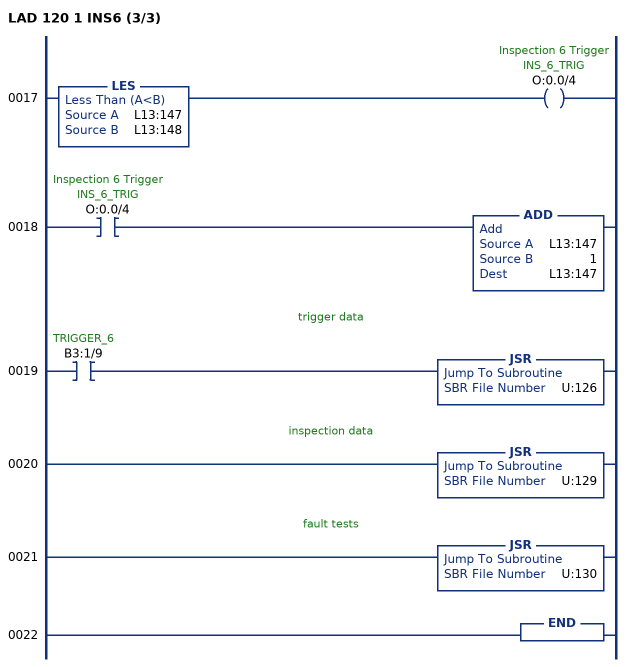
% Rung: 17 %
SOR LES L13:147 L13:148 OTE O:0.0/4 EOR
%   O:0.0/4  INS_6_TRIG  "Inspection 6 Trigger" %
% Rung: 18 %
SOR XIC O:0.0/4 ADD L13:147 1 L13:147 EOR
%   O:0.0/4  INS_6_TRIG  "Inspection 6 Trigger" %
% Rung: 19 %
% trigger data %
SOR XIC B3:1/9 JSR U:126 EOR
%   B3:1/9  TRIGGER_6 %
% Rung: 20 %
% inspection data %
SOR JSR U:129 EOR
% Rung: 21 %
% fault tests %
SOR JSR U:130 EOR
% Rung: 22 %
SOR END EOR

LADDER 121 "2 INS6RESU"
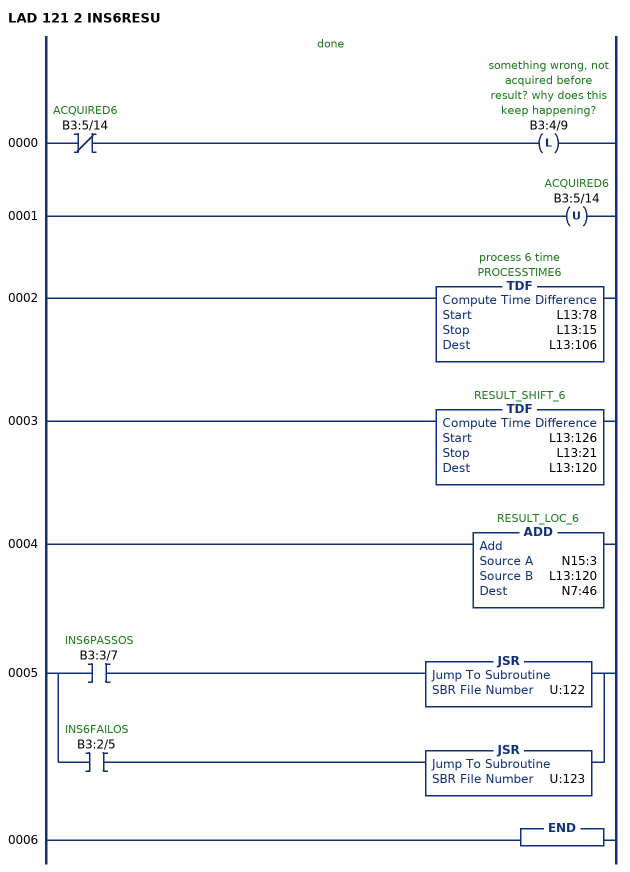
% Rung: 0 %
% done %
SOR XIO B3:5/14 OTL B3:4/9 EOR
%   B3:5/14  ACQUIRED6 %
%   B3:4/9  "something wrong, not acquired before result? why does this keep happening?" %
% Rung: 1 %
SOR OTU B3:5/14 EOR
%   B3:5/14  ACQUIRED6 %
% Rung: 2 %
SOR TDF L13:78 L13:15 L13:106 EOR
%   L13:78  TIMEOFACQ6  "the time of the last acquire" %
%   L13:15  THE_TIME %
%   L13:106  PROCESSTIME6  "process 6 time" %
% Rung: 3 %
SOR TDF L13:126 L13:21 L13:120 EOR
%   L13:126  PROCESS_START_POS_6 %
%   L13:21  TOP_POSITION %
%   L13:120  RESULT_SHIFT_6 %
% Rung: 4 %
SOR ADD N15:3 L13:120 N7:46 EOR
%   N15:3  INS_6_TRIG_LOC %
%   L13:120  RESULT_SHIFT_6 %
%   N7:46  RESULT_LOC_6 %
% Rung: 5 %
SOR BST XIC B3:3/7 JSR U:122 NXB XIC B3:2/5 JSR U:123 BND EOR
%   B3:3/7  INS6PASSOS %
%   B3:2/5  INS6FAILOS %
% Rung: 6 %
SOR END EOR

LADDER 122 "3 INS6PASS"
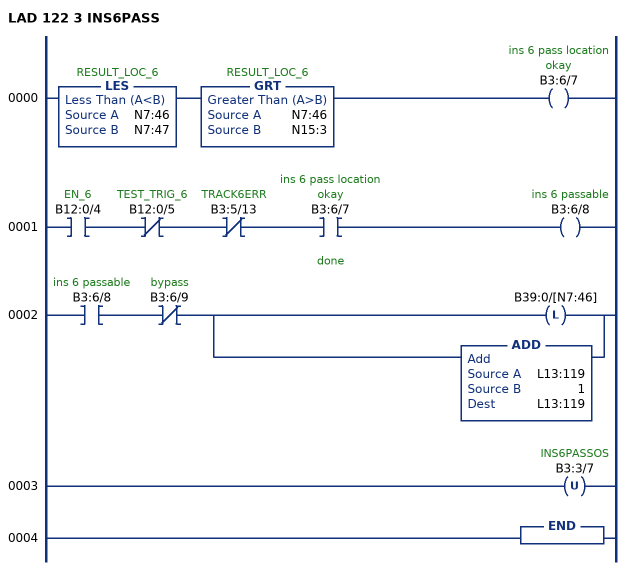
% Rung: 0 %
SOR LES N7:46 N7:47 GRT N7:46 N15:3 OTE B3:6/7 EOR
%   N7:46  RESULT_LOC_6 %
%   N7:47  INS6_MAX_SHIFT  "ins 6 maximum result location" %
%   N15:3  INS_6_TRIG_LOC %
%   B3:6/7  "ins 6 pass location okay" %
% Rung: 1 %
SOR XIC B12:0/4 XIO B12:0/5 XIO B3:5/13 XIC B3:6/7 OTE B3:6/8 EOR
%   B12:0/4  EN_6 %
%   B12:0/5  TEST_TRIG_6 %
%   B3:5/13  TRACK6ERR %
%   B3:6/7  "ins 6 pass location okay" %
%   B3:6/8  "ins 6 passable" %
% Rung: 2 %
% done %
SOR XIC B3:6/8 XIO B3:6/9 BST OTL B39:0/[N7:46] NXB ADD L13:119 1 L13:119 BND EOR
%   B3:6/8  "ins 6 passable" %
%   B3:6/9  "bypass" %
%   N7:46  RESULT_LOC_6 %
% Rung: 3 %
SOR OTU B3:3/7 EOR
%   B3:3/7  INS6PASSOS %
% Rung: 4 %
SOR END EOR

LADDER 123 "4 INS6FAIL"
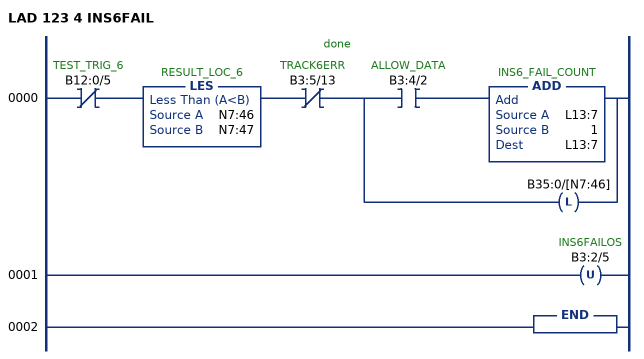
% Rung: 0 %
% done %
SOR XIO B12:0/5 LES N7:46 N7:47 XIO B3:5/13 BST XIC B3:4/2 ADD L13:7 1 L13:7 NXB OTL B35:0/[N7:46] BND EOR
%   B12:0/5  TEST_TRIG_6 %
%   N7:46  RESULT_LOC_6 %
%   N7:47  INS6_MAX_SHIFT  "ins 6 maximum result location" %
%   B3:5/13  TRACK6ERR %
%   B3:4/2  ALLOW_DATA %
%   L13:7  INS6_FAIL_COUNT %
%   B35:0  TOP_NG %
% Rung: 1 %
SOR OTU B3:2/5 EOR
%   B3:2/5  INS6FAILOS %
% Rung: 2 %
SOR END EOR

LADDER 124 "5 INS6ACQ"
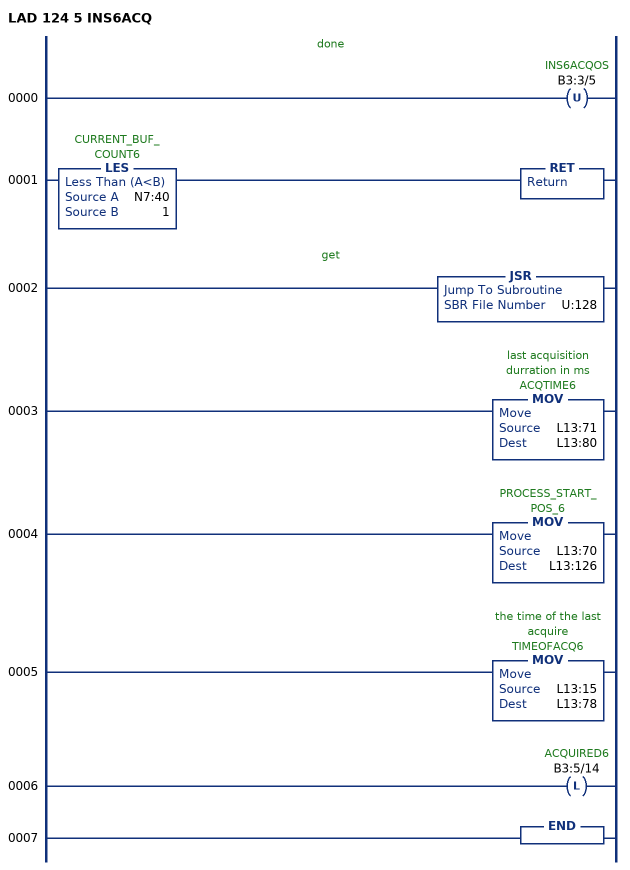
% Rung: 0 %
% done %
SOR OTU B3:3/5 EOR
%   B3:3/5  INS6ACQOS %
% Rung: 1 %
SOR LES N7:40 1 RET EOR
%   N7:40  CURRENT_BUF_COUNT6 %
% Rung: 2 %
% get %
SOR JSR U:128 EOR
% Rung: 3 %
SOR MOV L13:71 L13:80 EOR
%   L13:71  TIME_SPAN6 %
%   L13:80  ACQTIME6  "last acquisition durration in ms" %
% Rung: 4 %
SOR MOV L13:70 L13:126 EOR
%   L13:70  PULLED_POSITION6 %
%   L13:126  PROCESS_START_POS_6 %
% Rung: 5 %
SOR MOV L13:15 L13:78 EOR
%   L13:15  THE_TIME %
%   L13:78  TIMEOFACQ6  "the time of the last acquire" %
% Rung: 6 %
SOR OTL B3:5/14 EOR
%   B3:5/14  ACQUIRED6 %
% Rung: 7 %
SOR END EOR

LADDER 125 "6 Q6TESTTR"
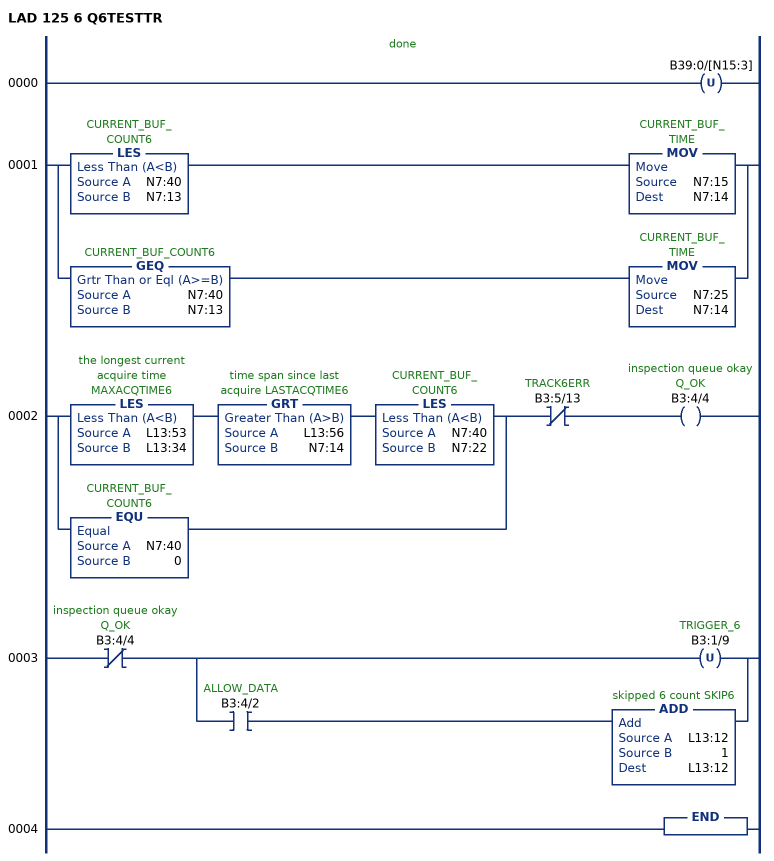
% Rung: 0 %
% done %
SOR OTU B39:0/[N15:3] EOR
%   N15:3  INS_6_TRIG_LOC %
% Rung: 1 %
SOR BST LES N7:40 N7:13 MOV N7:15 N7:14 NXB GEQ N7:40 N7:13 MOV N7:25 N7:14 BND EOR
%   N7:40  CURRENT_BUF_COUNT6 %
%   N7:13  BUF_TRANS  "cam to pc buf transition" %
%   N7:15  CAM_BUF_TIME  "cam buf time" %
%   N7:14  CURRENT_BUF_TIME %
%   N7:25  PC_BUF_TIME  "pc buf time" %
% Rung: 2 %
SOR BST LES L13:53 L13:34 GRT L13:56 N7:14 LES N7:40 N7:22 NXB EQU N7:40 0 BND XIO B3:5/13 OTE B3:4/4 EOR
%   L13:53  MAXACQTIME6  "the longest current acquire time" %
%   L13:34  MAX_ACQ_ALL  "absolute max acquire time before bypass trigger" %
%   L13:56  LASTACQTIME6  "time span since last acquire" %
%   N7:14  CURRENT_BUF_TIME %
%   N7:40  CURRENT_BUF_COUNT6 %
%   N7:22  MAX_BUF_ALL  "max buffer count alowed before bypass" %
%   B3:5/13  TRACK6ERR %
%   B3:4/4  Q_OK  "inspection queue okay" %
% Rung: 3 %
SOR XIO B3:4/4 BST OTU B3:1/9 NXB XIC B3:4/2 ADD L13:12 1 L13:12 BND EOR
%   B3:4/4  Q_OK  "inspection queue okay" %
%   B3:1/9  TRIGGER_6 %
%   B3:4/2  ALLOW_DATA %
%   L13:12  SKIP6  "skipped 6 count" %
% Rung: 4 %
SOR END EOR

LADDER 126 "7 INS6TRIG"
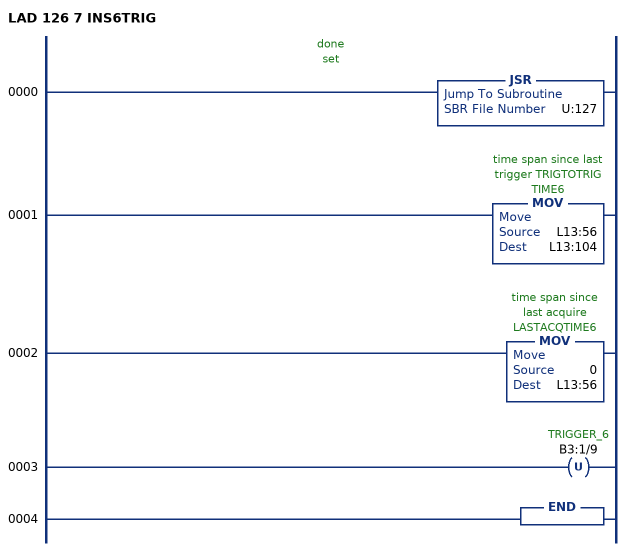
% Rung: 0 %
% done
% set %
SOR JSR U:127 EOR
% Rung: 1 %
SOR MOV L13:56 L13:104 EOR
%   L13:56  LASTACQTIME6  "time span since last acquire" %
%   L13:104  TRIGTOTRIGTIME6  "time span since last trigger" %
% Rung: 2 %
SOR MOV 0 L13:56 EOR
%   L13:56  LASTACQTIME6  "time span since last acquire" %
% Rung: 3 %
SOR OTU B3:1/9 EOR
%   B3:1/9  TRIGGER_6 %
% Rung: 4 %
SOR END EOR

LADDER 127 "8 FIFO6SET"
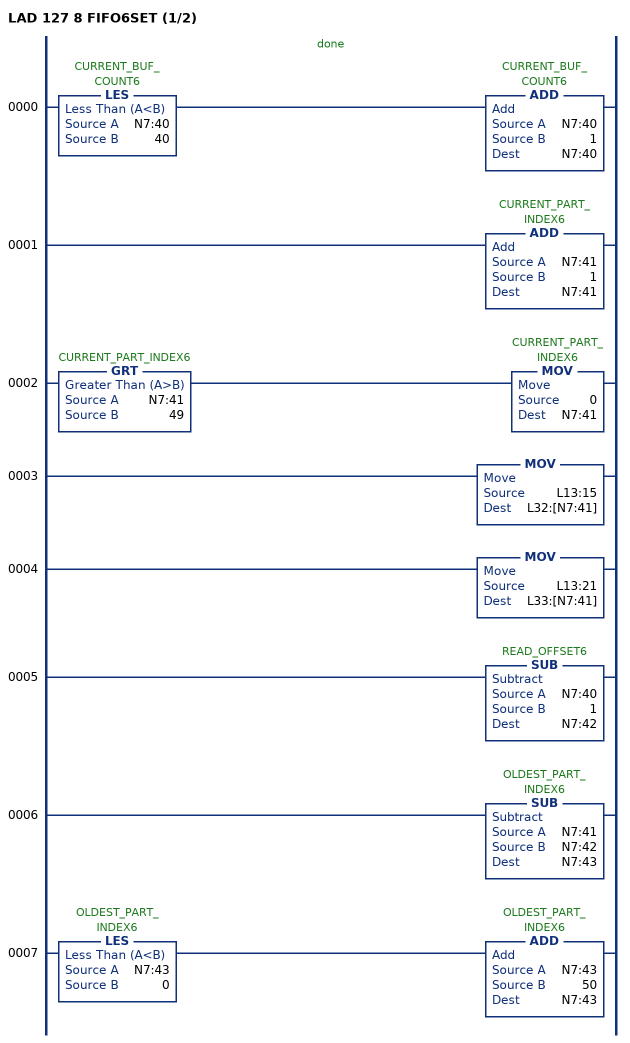
% Rung: 0 %
% done %
SOR LES N7:40 40 ADD N7:40 1 N7:40 EOR
%   N7:40  CURRENT_BUF_COUNT6 %
% Rung: 1 %
SOR ADD N7:41 1 N7:41 EOR
%   N7:41  CURRENT_PART_INDEX6 %
% Rung: 2 %
SOR GRT N7:41 49 MOV 0 N7:41 EOR
%   N7:41  CURRENT_PART_INDEX6 %
% Rung: 3 %
SOR MOV L13:15 L32:[N7:41] EOR
%   L13:15  THE_TIME %
%   N7:41  CURRENT_PART_INDEX6 %
% Rung: 4 %
SOR MOV L13:21 L33:[N7:41] EOR
%   L13:21  TOP_POSITION %
%   N7:41  CURRENT_PART_INDEX6 %
% Rung: 5 %
SOR SUB N7:40 1 N7:42 EOR
%   N7:40  CURRENT_BUF_COUNT6 %
%   N7:42  READ_OFFSET6 %
% Rung: 6 %
SOR SUB N7:41 N7:42 N7:43 EOR
%   N7:41  CURRENT_PART_INDEX6 %
%   N7:42  READ_OFFSET6 %
%   N7:43  OLDEST_PART_INDEX6 %
% Rung: 7 %
SOR LES N7:43 0 ADD N7:43 50 N7:43 EOR
%   N7:43  OLDEST_PART_INDEX6 %

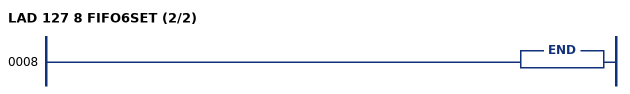
% Rung: 8 %
SOR END EOR

LADDER 128 "9 FIFO6GET"
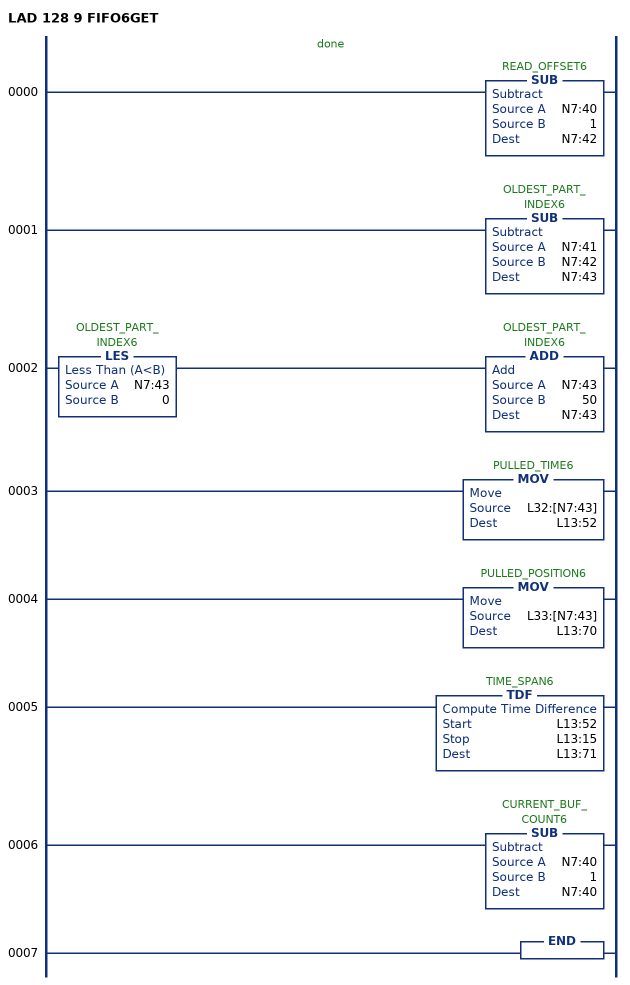
% Rung: 0 %
% done %
SOR SUB N7:40 1 N7:42 EOR
%   N7:40  CURRENT_BUF_COUNT6 %
%   N7:42  READ_OFFSET6 %
% Rung: 1 %
SOR SUB N7:41 N7:42 N7:43 EOR
%   N7:41  CURRENT_PART_INDEX6 %
%   N7:42  READ_OFFSET6 %
%   N7:43  OLDEST_PART_INDEX6 %
% Rung: 2 %
SOR LES N7:43 0 ADD N7:43 50 N7:43 EOR
%   N7:43  OLDEST_PART_INDEX6 %
% Rung: 3 %
SOR MOV L32:[N7:43] L13:52 EOR
%   N7:43  OLDEST_PART_INDEX6 %
%   L13:52  PULLED_TIME6 %
% Rung: 4 %
SOR MOV L33:[N7:43] L13:70 EOR
%   N7:43  OLDEST_PART_INDEX6 %
%   L13:70  PULLED_POSITION6 %
% Rung: 5 %
SOR TDF L13:52 L13:15 L13:71 EOR
%   L13:52  PULLED_TIME6 %
%   L13:15  THE_TIME %
%   L13:71  TIME_SPAN6 %
% Rung: 6 %
SOR SUB N7:40 1 N7:40 EOR
%   N7:40  CURRENT_BUF_COUNT6 %
% Rung: 7 %
SOR END EOR

LADDER 129 "10INSDATA6"
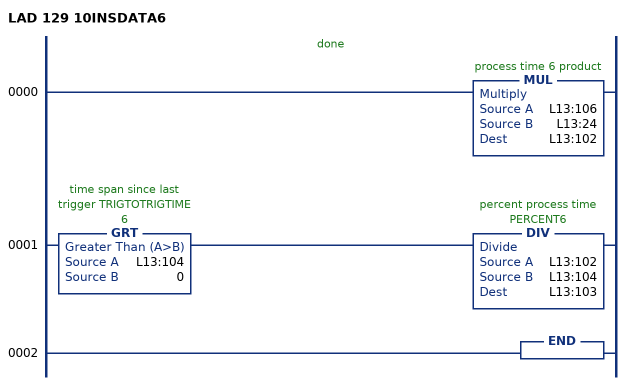
% Rung: 0 %
% done %
SOR MUL L13:106 L13:24 L13:102 EOR
%   L13:106  PROCESSTIME6  "process 6 time" %
%   L13:24  "multiplyer to make devision come out to a percentage" %
%   L13:102  "process time 6 product" %
% Rung: 1 %
SOR GRT L13:104 0 DIV L13:102 L13:104 L13:103 EOR
%   L13:104  TRIGTOTRIGTIME6  "time span since last trigger" %
%   L13:102  "process time 6 product" %
%   L13:103  PERCENT6  "percent process time" %
% Rung: 2 %
SOR END EOR

LADDER 130 "11TSTFALT6"
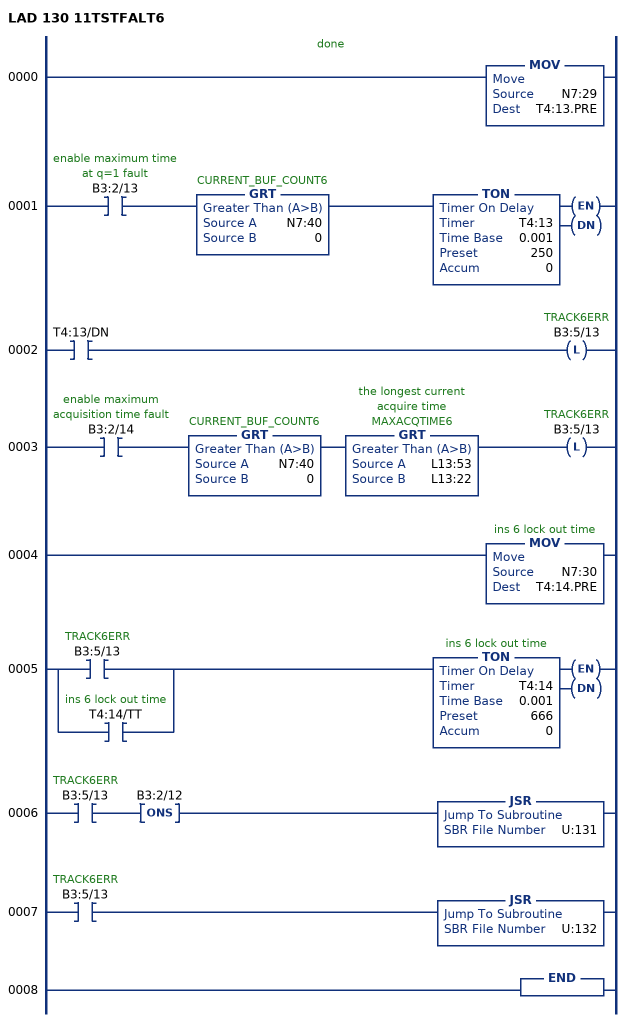
% Rung: 0 %
% done %
SOR MOV N7:29 T4:13.PRE EOR
%   N7:29  "max allowed ms time for q to be above 1 if safe fault is used" %
% Rung: 1 %
SOR XIC B3:2/13 GRT N7:40 0 TON T4:13 0.001 250 0 EOR
%   B3:2/13  "enable maximum time at q=1 fault" %
%   N7:40  CURRENT_BUF_COUNT6 %
% Rung: 2 %
SOR XIC T4:13/DN OTL B3:5/13 EOR
%   B3:5/13  TRACK6ERR %
% Rung: 3 %
SOR XIC B3:2/14 GRT N7:40 0 GRT L13:53 L13:22 OTL B3:5/13 EOR
%   B3:2/14  "enable maximum acquisition time fault" %
%   N7:40  CURRENT_BUF_COUNT6 %
%   L13:53  MAXACQTIME6  "the longest current acquire time" %
%   L13:22  "maximum of the longest acquire time allowed if maximum acquire time fault is enabled" %
%   B3:5/13  TRACK6ERR %
% Rung: 4 %
SOR MOV N7:30 T4:14.PRE EOR
%   N7:30  "ms time setting to lock out inspection to give all pending images a chance to clear" %
%   T4:14  "ins 6 lock out time" %
% Rung: 5 %
SOR BST XIC B3:5/13 NXB XIC T4:14/TT BND TON T4:14 0.001 666 0 EOR
%   B3:5/13  TRACK6ERR %
%   T4:14  "ins 6 lock out time" %
% Rung: 6 %
SOR XIC B3:5/13 ONS B3:2/12 JSR U:131 EOR
%   B3:5/13  TRACK6ERR %
% Rung: 7 %
SOR XIC B3:5/13 JSR U:132 EOR
%   B3:5/13  TRACK6ERR %
% Rung: 8 %
SOR END EOR

LADDER 131 "12INS6FIX1"
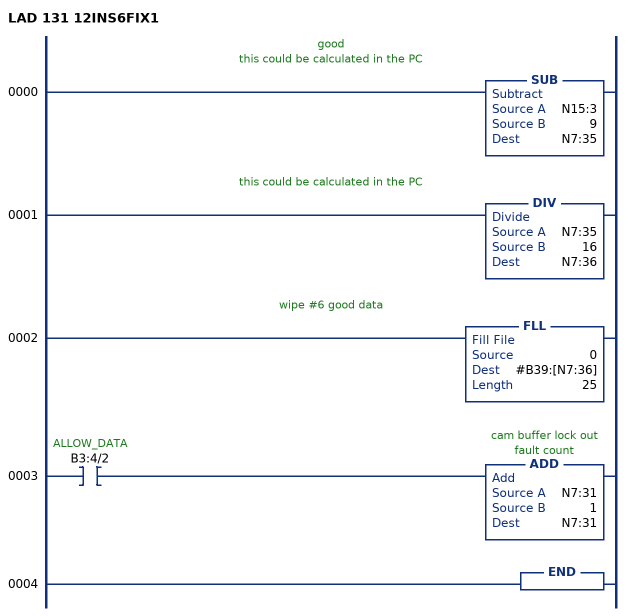
% Rung: 0 %
% good
% this could be calculated in the PC %
SOR SUB N15:3 9 N7:35 EOR
%   N15:3  INS_6_TRIG_LOC %
% Rung: 1 %
% this could be calculated in the PC %
SOR DIV N7:35 16 N7:36 EOR
% Rung: 2 %
% wipe #6 good data %
SOR FLL 0 #B39:[N7:36] 25 EOR
% Rung: 3 %
SOR XIC B3:4/2 ADD N7:31 1 N7:31 EOR
%   B3:4/2  ALLOW_DATA %
%   N7:31  "cam buffer lock out fault count" %
% Rung: 4 %
SOR END EOR

LADDER 132 "13INS6FIX2"
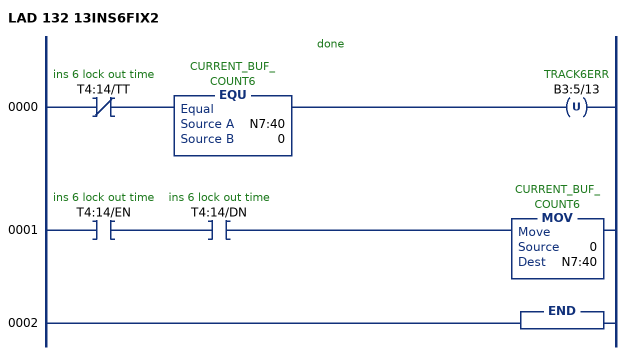
% Rung: 0 %
% done %
SOR XIO T4:14/TT EQU N7:40 0 OTU B3:5/13 EOR
%   T4:14  "ins 6 lock out time" %
%   N7:40  CURRENT_BUF_COUNT6 %
%   B3:5/13  TRACK6ERR %
% Rung: 1 %
SOR XIC T4:14/EN XIC T4:14/DN MOV 0 N7:40 EOR
%   T4:14  "ins 6 lock out time" %
%   N7:40  CURRENT_BUF_COUNT6 %
% Rung: 2 %
SOR END EOR

LADDER 133 "14 HSTRIG6"
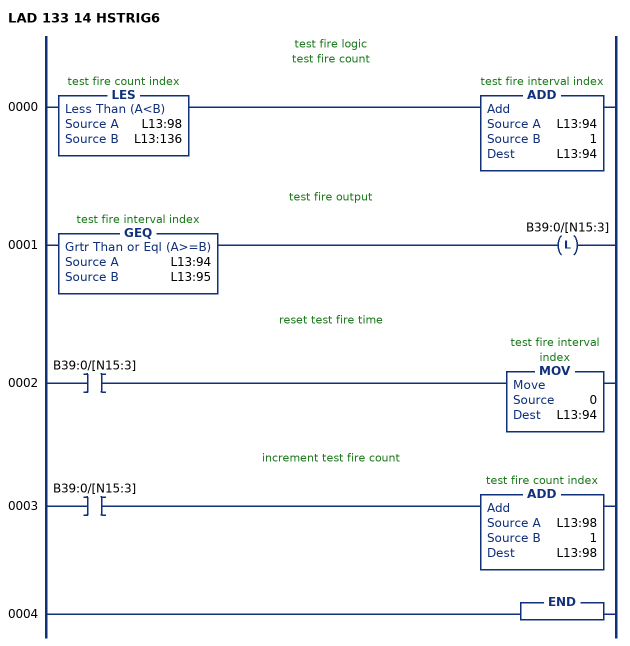
% Rung: 0 %
% test fire logic
% 
% test fire count %
SOR LES L13:98 L13:136 ADD L13:94 1 L13:94 EOR
%   L13:98  "test fire count index" %
%   L13:136  "test fire count" %
%   L13:94  "test fire interval index" %
% Rung: 1 %
% test fire output %
SOR GEQ L13:94 L13:95 OTL B39:0/[N15:3] EOR
%   L13:94  "test fire interval index" %
%   L13:95  "test fire interval" %
%   N15:3  INS_6_TRIG_LOC %
% Rung: 2 %
% reset test fire time %
SOR XIC B39:0/[N15:3] MOV 0 L13:94 EOR
%   N15:3  INS_6_TRIG_LOC %
%   L13:94  "test fire interval index" %
% Rung: 3 %
% increment test fire count %
SOR XIC B39:0/[N15:3] ADD L13:98 1 L13:98 EOR
%   N15:3  INS_6_TRIG_LOC %
%   L13:98  "test fire count index" %
% Rung: 4 %
SOR END EOR

LADDER 190 "PASS BLOW"
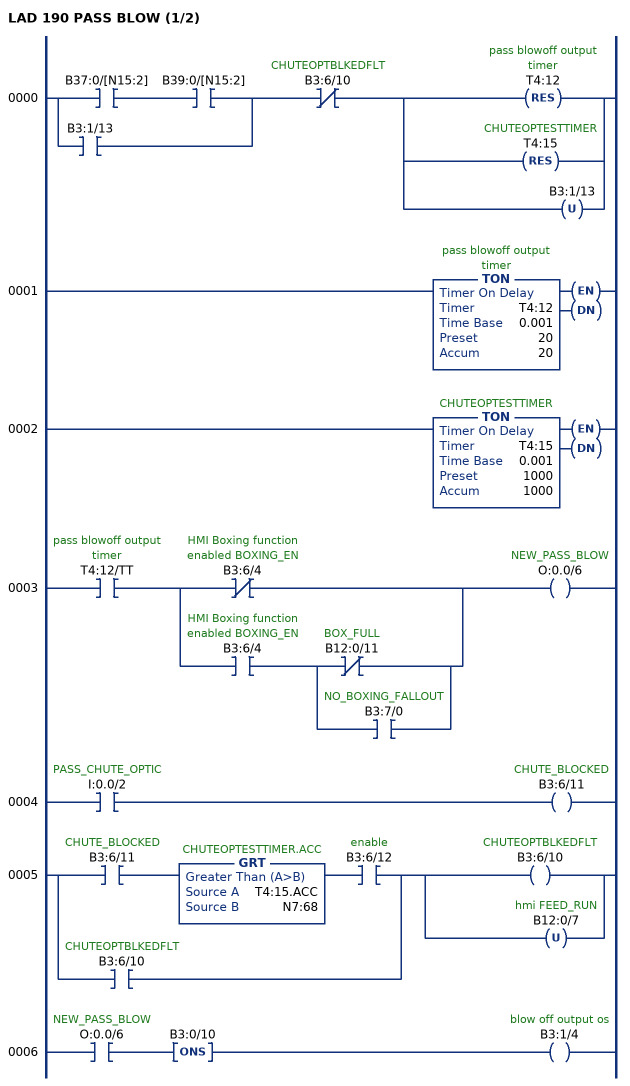
% Rung: 0 %
SOR BST XIC B37:0/[N15:2] XIC B39:0/[N15:2] NXB XIC B3:1/13 BND XIO B3:6/10 BST RES T4:12 NXB RES T4:15 NXB OTU B3:1/13 BND EOR
%   N15:2  BLOW_PT %
%   B3:6/10  CHUTEOPTBLKEDFLT %
%   T4:12  "pass blowoff output timer" %
%   T4:15  CHUTEOPTESTTIMER %
% Rung: 1 %
SOR TON T4:12 0.001 20 20 EOR
%   T4:12  "pass blowoff output timer" %
% Rung: 2 %
SOR TON T4:15 0.001 1000 1000 EOR
%   T4:15  CHUTEOPTESTTIMER %
% Rung: 3 %
SOR XIC T4:12/TT BST XIO B3:6/4 NXB XIC B3:6/4 BST XIO B12:0/11 NXB XIC B3:7/0 BND BND OTE O:0.0/6 EOR
%   T4:12  "pass blowoff output timer" %
%   B3:6/4  BOXING_EN  "HMI Boxing function enabled" %
%   B12:0/11  BOX_FULL %
%   B3:7/0  NO_BOXING_FALLOUT %
%   O:0.0/6  NEW_PASS_BLOW %
% Rung: 4 %
SOR XIC I:0.0/2 OTE B3:6/11 EOR
%   I:0.0/2  PASS_CHUTE_OPTIC %
%   B3:6/11  CHUTE_BLOCKED %
% Rung: 5 %
SOR BST XIC B3:6/11 GRT T4:15.ACC N7:68 XIC B3:6/12 NXB XIC B3:6/10 BND BST OTE B3:6/10 NXB OTU B12:0/7 BND EOR
%   B3:6/11  CHUTE_BLOCKED %
%   T4:15  CHUTEOPTESTTIMER %
%   B3:6/12  "enable" %
%   B3:6/10  CHUTEOPTBLKEDFLT %
%   B12:0/7  FEED_RUN  "hmi" %
% Rung: 6 %
SOR XIC O:0.0/6 ONS B3:0/10 OTE B3:1/4 EOR
%   O:0.0/6  NEW_PASS_BLOW %
%   B3:1/4  "blow off output os" %

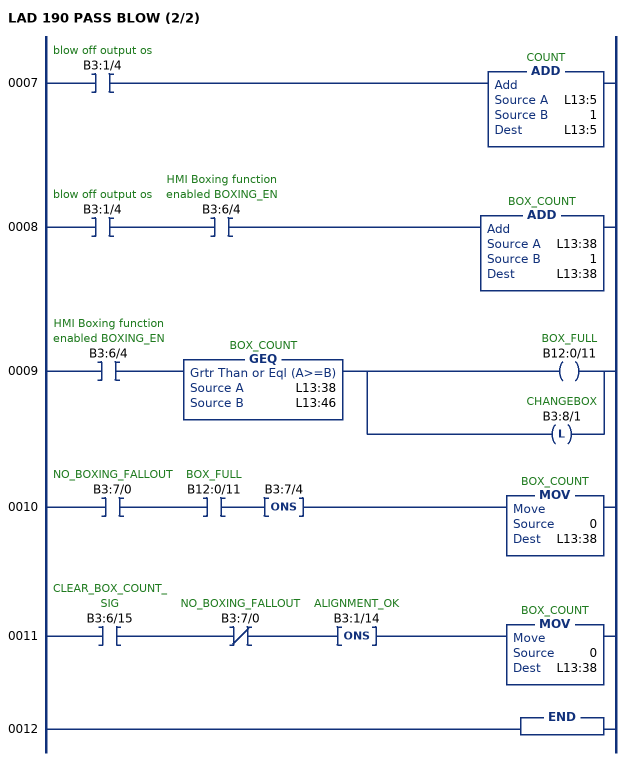
% Rung: 7 %
SOR XIC B3:1/4 ADD L13:5 1 L13:5 EOR
%   B3:1/4  "blow off output os" %
%   L13:5  COUNT %
% Rung: 8 %
SOR XIC B3:1/4 XIC B3:6/4 ADD L13:38 1 L13:38 EOR
%   B3:1/4  "blow off output os" %
%   B3:6/4  BOXING_EN  "HMI Boxing function enabled" %
%   L13:38  BOX_COUNT %
% Rung: 9 %
SOR XIC B3:6/4 GEQ L13:38 L13:46 BST OTE B12:0/11 NXB OTL B3:8/1 BND EOR
%   B3:6/4  BOXING_EN  "HMI Boxing function enabled" %
%   L13:38  BOX_COUNT %
%   L13:46  BOX_LIMIT  "box count setpoint" %
%   B12:0/11  BOX_FULL %
%   B3:8/1  CHANGEBOX %
% Rung: 10 %
SOR XIC B3:7/0 XIC B12:0/11 ONS B3:7/4 MOV 0 L13:38 EOR
%   B3:7/0  NO_BOXING_FALLOUT %
%   B12:0/11  BOX_FULL %
%   L13:38  BOX_COUNT %
% Rung: 11 %
SOR XIC B3:6/15 XIO B3:7/0 ONS B3:1/14 MOV 0 L13:38 EOR
%   B3:6/15  CLEAR_BOX_COUNT_SIG %
%   B3:7/0  NO_BOXING_FALLOUT %
%   B3:1/14  ALIGNMENT_OK %
%   L13:38  BOX_COUNT %
% Rung: 12 %
SOR END EOR

LADDER 201 "UNUSED"
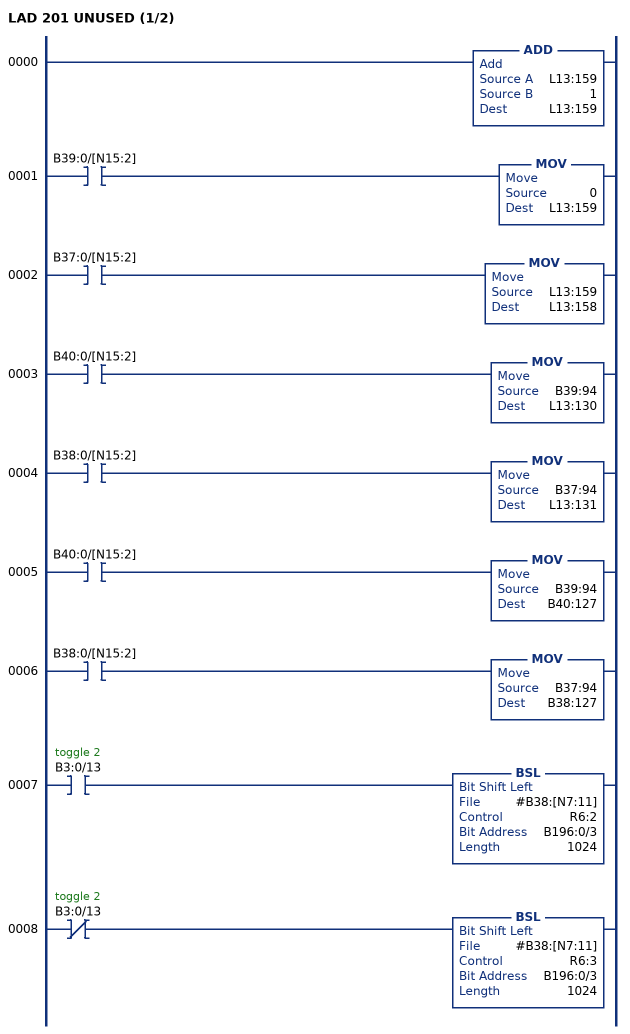
% Rung: 0 %
SOR ADD L13:159 1 L13:159 EOR
% Rung: 1 %
SOR XIC B39:0/[N15:2] MOV 0 L13:159 EOR
%   N15:2  BLOW_PT %
% Rung: 2 %
SOR XIC B37:0/[N15:2] MOV L13:159 L13:158 EOR
%   N15:2  BLOW_PT %
% Rung: 3 %
SOR XIC B40:0/[N15:2] MOV B39:94 L13:130 EOR
%   N15:2  BLOW_PT %
% Rung: 4 %
SOR XIC B38:0/[N15:2] MOV B37:94 L13:131 EOR
%   N15:2  BLOW_PT %
% Rung: 5 %
SOR XIC B40:0/[N15:2] MOV B39:94 B40:127 EOR
%   N15:2  BLOW_PT %
% Rung: 6 %
SOR XIC B38:0/[N15:2] MOV B37:94 B38:127 EOR
%   N15:2  BLOW_PT %
% Rung: 7 %
SOR XIC B3:0/13 BSL #B38:[N7:11] R6:2 B196:0/3 1024 EOR
%   B3:0/13  "toggle 2" %
%   B196:0/3  OFF %
% Rung: 8 %
SOR XIO B3:0/13 BSL #B38:[N7:11] R6:3 B196:0/3 1024 EOR
%   B3:0/13  "toggle 2" %
%   B196:0/3  OFF %

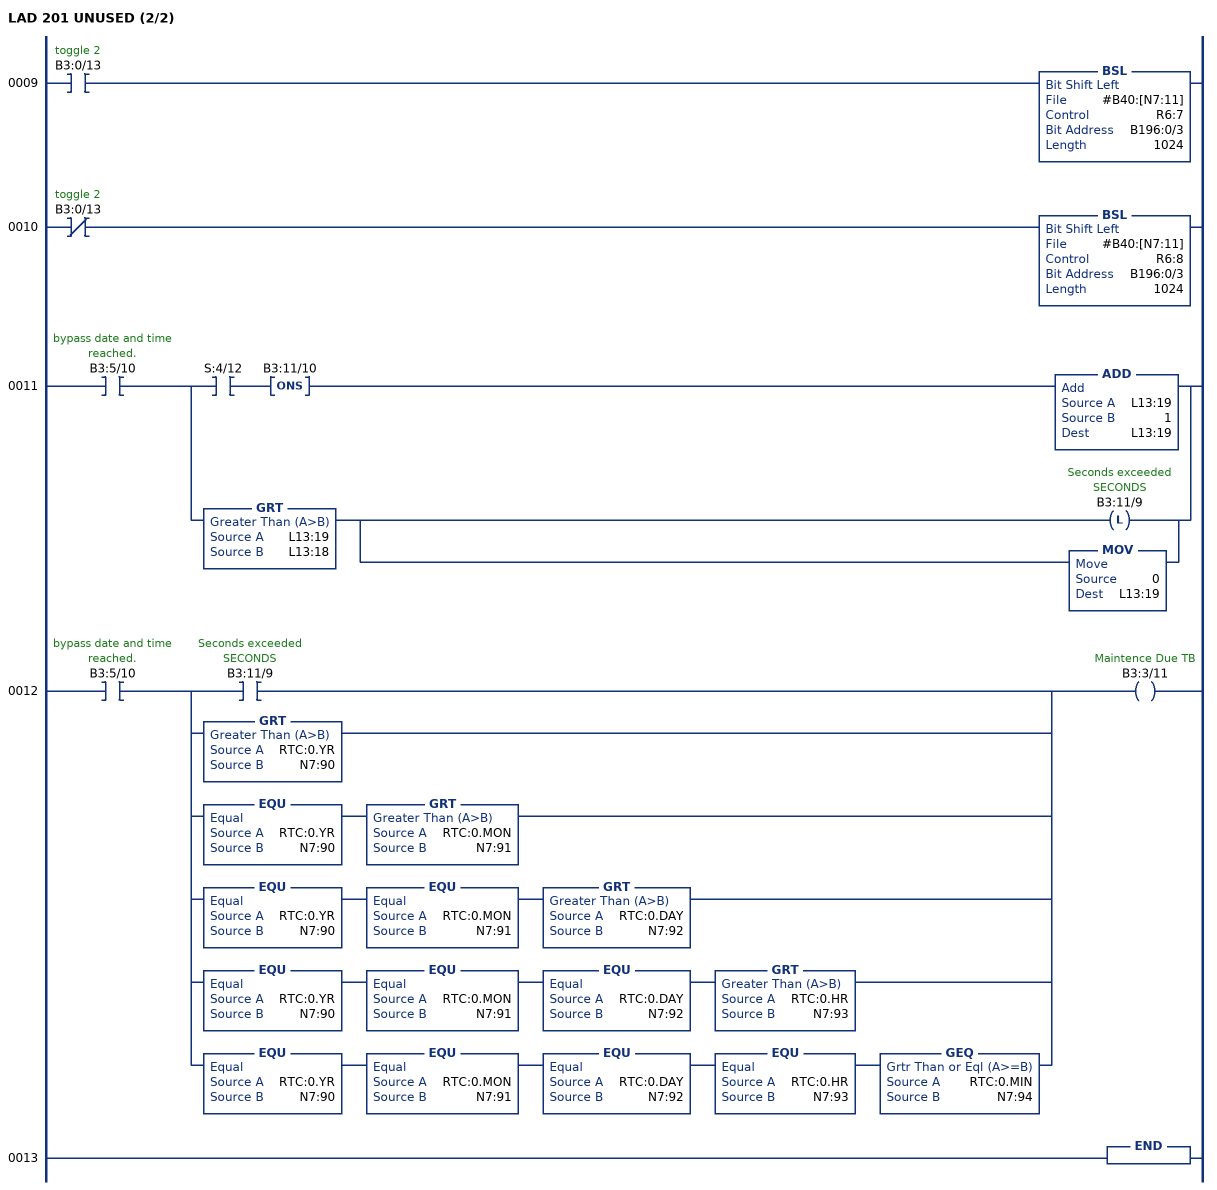
% Rung: 9 %
SOR XIC B3:0/13 BSL #B40:[N7:11] R6:7 B196:0/3 1024 EOR
%   B3:0/13  "toggle 2" %
%   B196:0/3  OFF %
% Rung: 10 %
SOR XIO B3:0/13 BSL #B40:[N7:11] R6:8 B196:0/3 1024 EOR
%   B3:0/13  "toggle 2" %
%   B196:0/3  OFF %
% Rung: 11 %
SOR XIC B3:5/10 BST XIC S:4/12 ONS B3:11/10 ADD L13:19 1 L13:19 NXB GRT L13:19 L13:18 BST OTL B3:11/9 NXB MOV 0 L13:19 BND BND EOR
%   B3:5/10  "bypass date and time reached." %
%   L13:18  MAX %
%   B3:11/9  SECONDS  "Seconds exceeded" %
% Rung: 12 %
SOR XIC B3:5/10 BST XIC B3:11/9 NXB GRT RTC:0.YR N7:90 NXB EQU RTC:0.YR N7:90 GRT RTC:0.MON N7:91 NXB EQU RTC:0.YR N7:90 EQU RTC:0.MON N7:91 GRT RTC:0.DAY N7:92 NXB EQU RTC:0.YR N7:90 EQU RTC:0.MON N7:91 EQU RTC:0.DAY N7:92 GRT RTC:0.HR N7:93 NXB EQU RTC:0.YR N7:90 EQU RTC:0.MON N7:91 EQU RTC:0.DAY N7:92 EQU RTC:0.HR N7:93 GEQ RTC:0.MIN N7:94 BND OTE B3:3/11 EOR
%   B3:5/10  "bypass date and time reached." %
%   B3:11/9  SECONDS  "Seconds exceeded" %
%   N7:90  RTC %
%   B3:3/11  TB  "Maintence Due" %
% Rung: 13 %
SOR END EOR

LADDER 215 "TESTTRIG1"
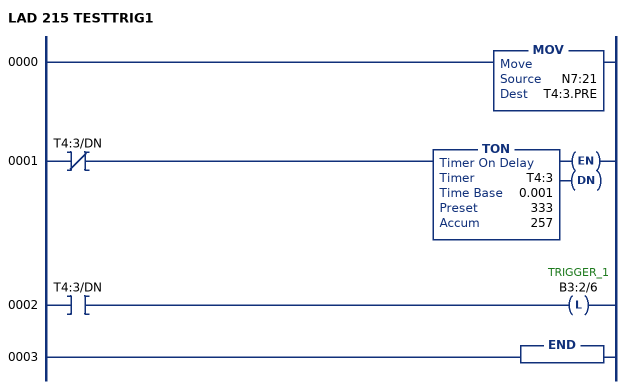
% Rung: 0 %
SOR MOV N7:21 T4:3.PRE EOR
% Rung: 1 %
SOR XIO T4:3/DN TON T4:3 0.001 333 257 EOR
% Rung: 2 %
SOR XIC T4:3/DN OTL B3:2/6 EOR
%   B3:2/6  TRIGGER_1 %
% Rung: 3 %
SOR END EOR

LADDER 216 "TESTTRIG5"
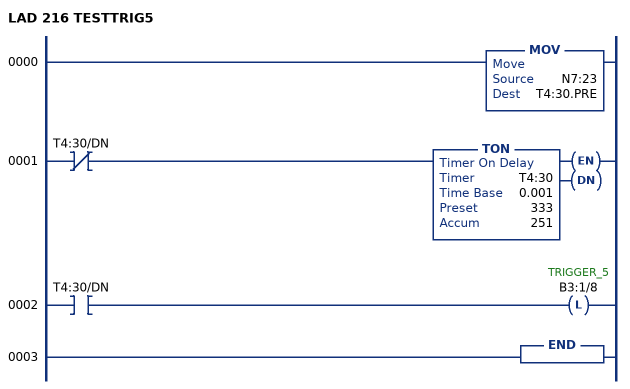
% Rung: 0 %
SOR MOV N7:23 T4:30.PRE EOR
% Rung: 1 %
SOR XIO T4:30/DN TON T4:30 0.001 333 251 EOR
% Rung: 2 %
SOR XIC T4:30/DN OTL B3:1/8 EOR
%   B3:1/8  TRIGGER_5 %
% Rung: 3 %
SOR END EOR

LADDER 217 "TESTTRIG6"
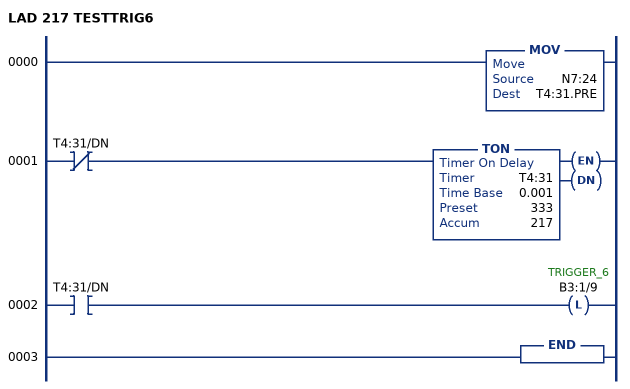
% Rung: 0 %
SOR MOV N7:24 T4:31.PRE EOR
% Rung: 1 %
SOR XIO T4:31/DN TON T4:31 0.001 333 217 EOR
% Rung: 2 %
SOR XIC T4:31/DN OTL B3:1/9 EOR
%   B3:1/9  TRIGGER_6 %
% Rung: 3 %
SOR END EOR

LADDER 219 "PACKAGER"    % normal %
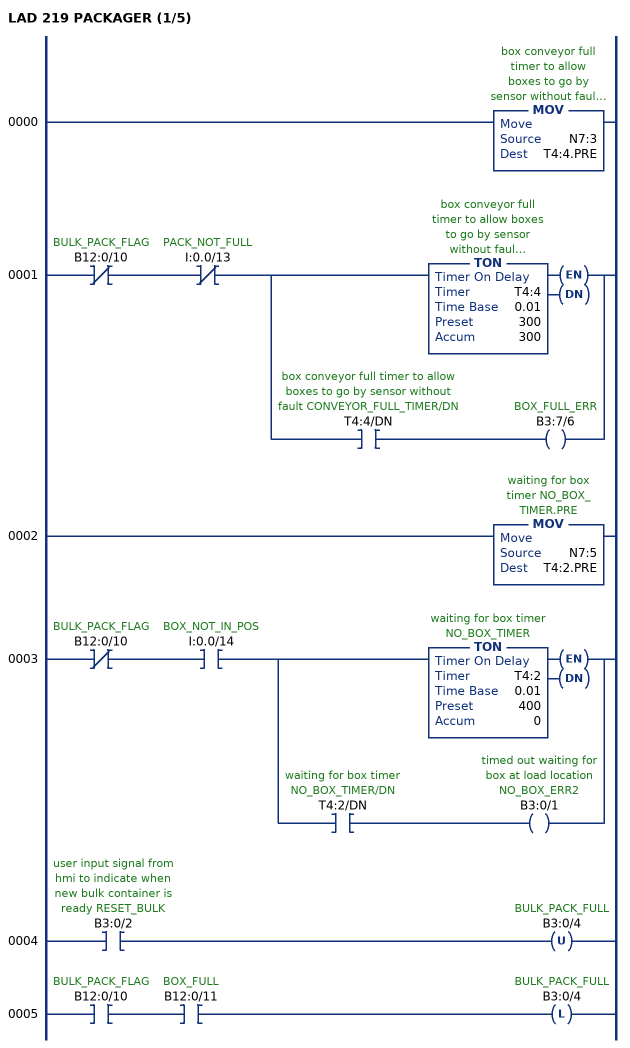
% Rung: 0 %
SOR MOV N7:3 T4:4.PRE EOR
%   N7:3  "time to allow box to pass box conveyor full sensor without fault" %
%   T4:4  CONVEYOR_FULL_TIMER  "box conveyor full timer to allow boxes to go by sensor without fault" %
% Rung: 1 %
SOR XIO B12:0/10 XIO I:0.0/13 BST TON T4:4 0.01 300 300 NXB XIC T4:4/DN OTE B3:7/6 BND EOR
%   B12:0/10  BULK_PACK_FLAG %
%   I:0.0/13  PACK_NOT_FULL %
%   T4:4  CONVEYOR_FULL_TIMER  "box conveyor full timer to allow boxes to go by sensor without fault" %
%   B3:7/6  BOX_FULL_ERR %
% Rung: 2 %
SOR MOV N7:5 T4:2.PRE EOR
%   N7:5  "buffer count 6" %
%   T4:2  NO_BOX_TIMER  "waiting for box timer" %
% Rung: 3 %
SOR XIO B12:0/10 XIC I:0.0/14 BST TON T4:2 0.01 400 0 NXB XIC T4:2/DN OTE B3:0/1 BND EOR
%   B12:0/10  BULK_PACK_FLAG %
%   I:0.0/14  BOX_NOT_IN_POS %
%   T4:2  NO_BOX_TIMER  "waiting for box timer" %
%   B3:0/1  NO_BOX_ERR2  "timed out waiting for box at load location" %
% Rung: 4 %
SOR XIC B3:0/2 OTU B3:0/4 EOR
%   B3:0/2  RESET_BULK  "user input signal from hmi to indicate when new bulk container is ready" %
%   B3:0/4  BULK_PACK_FULL %
% Rung: 5 %
SOR XIC B12:0/10 XIC B12:0/11 OTL B3:0/4 EOR
%   B12:0/10  BULK_PACK_FLAG %
%   B12:0/11  BOX_FULL %
%   B3:0/4  BULK_PACK_FULL %

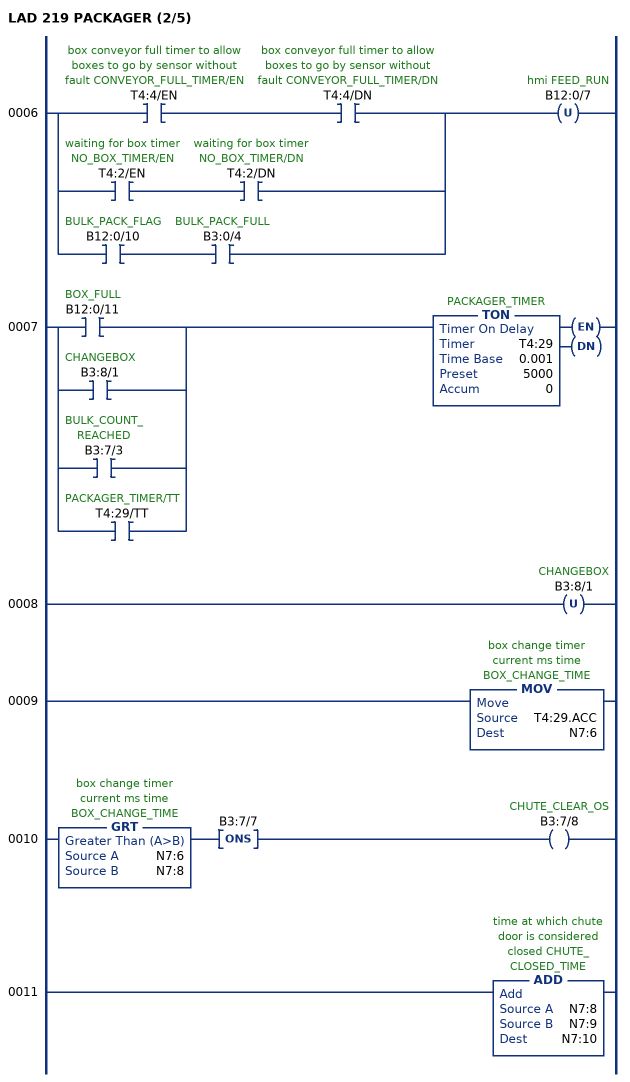
% Rung: 6 %
SOR BST XIC T4:4/EN XIC T4:4/DN NXB XIC T4:2/EN XIC T4:2/DN NXB XIC B12:0/10 XIC B3:0/4 BND OTU B12:0/7 EOR
%   T4:4  CONVEYOR_FULL_TIMER  "box conveyor full timer to allow boxes to go by sensor without fault" %
%   T4:2  NO_BOX_TIMER  "waiting for box timer" %
%   B12:0/10  BULK_PACK_FLAG %
%   B3:0/4  BULK_PACK_FULL %
%   B12:0/7  FEED_RUN  "hmi" %
% Rung: 7 %
SOR BST XIC B12:0/11 NXB XIC B3:8/1 NXB XIC B3:7/3 NXB XIC T4:29/TT BND TON T4:29 0.001 5000 0 EOR
%   B12:0/11  BOX_FULL %
%   B3:8/1  CHANGEBOX %
%   B3:7/3  BULK_COUNT_REACHED %
%   T4:29  PACKAGER_TIMER %
% Rung: 8 %
SOR OTU B3:8/1 EOR
%   B3:8/1  CHANGEBOX %
% Rung: 9 %
SOR MOV T4:29.ACC N7:6 EOR
%   T4:29  PACKAGER_TIMER %
%   N7:6  BOX_CHANGE_TIME  "box change timer current ms time" %
% Rung: 10 %
SOR GRT N7:6 N7:8 ONS B3:7/7 OTE B3:7/8 EOR
%   N7:6  BOX_CHANGE_TIME  "box change timer current ms time" %
%   N7:8  CHUTE_CLEAR_TIME %
%   B3:7/8  CHUTE_CLEAR_OS %
% Rung: 11 %
SOR ADD N7:8 N7:9 N7:10 EOR
%   N7:8  CHUTE_CLEAR_TIME %
%   N7:9  CHUTE_CLOSE_TIME  "ms time required to close chute" %
%   N7:10  CHUTE_CLOSED_TIME  "time at which chute door is considered closed" %

